// TIA Portal V19 export
TYPE "lexchangetray_typeUnEmn_toConstraintWorkstationDeliver"
// Type: lexchangetray_typeUnEmn_toConstraintWorkstationReq
// Type: lexchangetray_typeUnEmn_toConstraintWorkstationFeedback
// stored: Access Published
   STRUCT
      feedback : "lexchangetray_typeUnEmn_toConstraintWorkstationFeedback";
      req : "lexchangetray_typeUnEmn_toConstraintWorkstationReq";
   END_STRUCT;
END_TYPE
